Fanuc KAREL source: kb00047.KL

PROGRAM KB00047
%STACKSIZE=65535
%PRIORITY=65535
%NOLOCKGROUP
VAR
P1 : STRING[80]
P2 : STRING[80]
P3 : BOOLEAN
P4 : INTEGER
BEGIN
P1='A'
P2='A'
P3=TRUE
P4=1
COPY_TPE(P1,P2,P3,P4)
END KB00047
